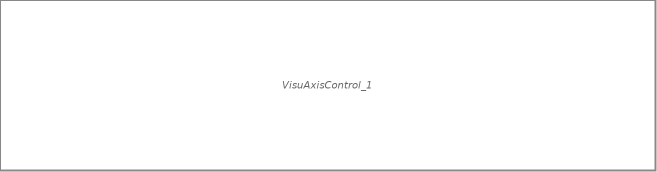
VISUALIZATION VisuAxisZ_1  // 657x172
    Frame (0,0 655x170)
        shows VisuAxisControl_1(sAxisName_1 := sAxisZName, stAxisVisu_1 := stAxisZ)
END_VISUALIZATION

(* stored: Version 1.1.0.1, ProductVersion 3.1.4022.6
   Visu VisuAxisZ_1: Id {1abdefd8-ad30-4da3-beb3-ef21682d5abb} *)
